// TIA Portal V18 export
DATA_BLOCK "L1_AssiAA"   // DB24
{ S7_Optimized_Access := 'TRUE' }
VERSION : 0.1
// stored: AutoNumber true, DBAccessibleFromOPCUA true, DBAccessibleFromWebserver true, IsOnlyStoredInLoadMemory false, IsRetainMemResEnabled false, IsWriteProtectedInAS false, MemoryReserve 100
   VAR RETAIN
      asse { S7_SetPoint := 'True'} : Array[1.."N_AssiAAA"] of "LGasp_typeAssiAAA";
   END_VAR
BEGIN
END_DATA_BLOCK
